FUNCTION_BLOCK DCAxis EXTENDS ParentAxis
VAR
END_VAR

METHOD StartDisable : BOOL
StartDisable := TRUE;
RETURN;
END_METHOD

METHOD StartEnable : BOOL
StartEnable := TRUE;
RETURN;
END_METHOD

METHOD StartErrorChecking : BOOL
StartErrorChecking := TRUE;
RETURN;
END_METHOD

METHOD StartMovement : BOOL
StartMovement := TRUE;
RETURN;
END_METHOD

METHOD StartReset : BOOL
StartReset := TRUE;
RETURN;
END_METHOD

END_FUNCTION_BLOCK

(* stored: Version 1.1.0.1, ProductVersion 3.1.4024.12
   POU DCAxis: Id {dea0db48-55b5-4854-89d4-e9ebef2095e4}, SpecialFunc None
   Folder METH: Id {e01e1756-1fa3-470d-8b52-d4b6bbbe0798}
   Folder PROP: Id {264c8613-12bc-4d33-9c4e-c9d79e1e4c31}
   Method StartDisable: Id {9cc790e2-ee6f-4695-94df-f544171a66ae}
   Method StartEnable: Id {c3cc6cf9-0720-4604-91cc-52924082bae0}
   Method StartErrorChecking: Id {b5fcf36a-71f5-4463-847d-7bd13b70b3b0}
   Method StartMovement: Id {853e969d-f18f-4abd-9e39-6f5c4ce4b98a}
   Method StartReset: Id {854ab7b6-9a61-47ad-84d0-ce102954eb45} *)
